SUBAPPLICATION SwitchPicCol_5_2 (* Bild- und Farbumschaltung für AUX-N und VT Objekte; 5 Zustände *)
  (* Standard: 61499-2 *)
  (* Version 1.1, 2026-04-09, Christoph Behr, HR Agrartechnik, Inits verbunden und REQ angeschlossen *)
  (* Version 1.0, 2025-06-12, franz, Meisterschulen am Ostbahnhof *)
  PACKAGE MyLib::sys;
  IMPORT logiBUS::utils::sequence::schieber::SchieberAuxInStruct;
  IMPORT logiBUS::utils::sequence::schieber::const::iSTATES::Unknown;
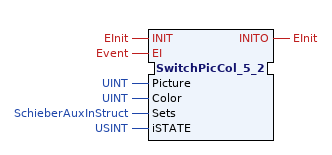
  EVENT_INPUT
    INIT : EInit; (* Initialization Request *)
    EI;
  END_EVENT
  EVENT_OUTPUT
    INITO : EInit; (* Initialization Confirm *)
  END_EVENT
  VAR_INPUT
    Picture : UINT; (* Object ID of the ObjectPointer to the Picture *)
    Color : UINT; (* Object ID of the AuxFunction *)
    Sets : logiBUS::utils::sequence::schieber::SchieberAuxInStruct;
    iSTATE : USINT := Unknown;
  END_VAR
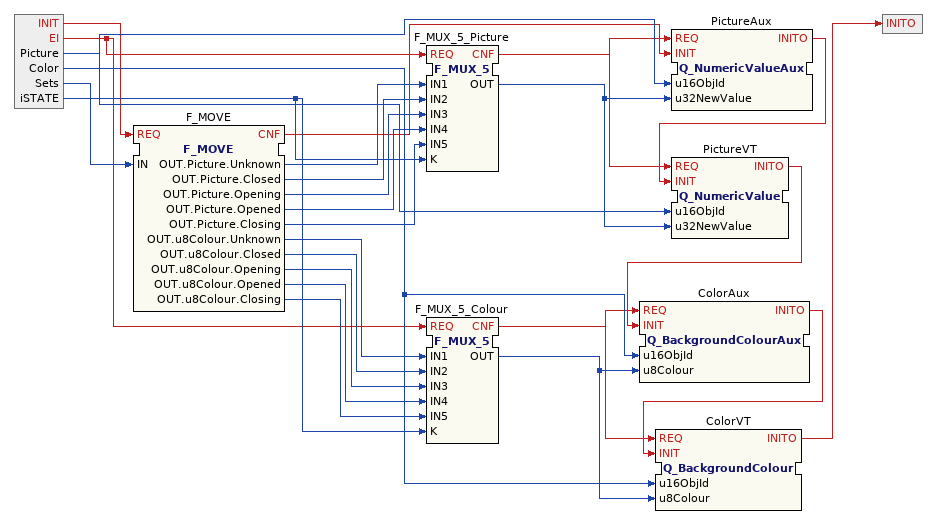
  FBS
    PictureVT : isobus::UT::Q::Q_NumericValue;
    ColorAux : isobus::UT::Q::Q_BackgroundColourAux;
    PictureAux : isobus::UT::Q::Q_NumericValueAux;
    ColorVT : isobus::UT::Q::Q_BackgroundColour;
    F_MOVE : iec61131::selection::F_MOVE; {SET_ATTRIBUTE(DataType, logiBUS::utils::sequence::schieber::SchieberAuxInStruct)}
    F_MUX_5_Picture : iec61131::selection::F_MUX_5;
    F_MUX_5_Colour : iec61131::selection::F_MUX_5;
  END_FBS
  EVENT_CONNECTIONS
    F_MUX_5_Picture.CNF TO PictureAux.REQ;
    F_MUX_5_Picture.CNF TO PictureVT.REQ;
    F_MUX_5_Colour.CNF TO ColorAux.REQ;
    F_MUX_5_Colour.CNF TO ColorVT.REQ;
    EI TO F_MUX_5_Picture.REQ;
    EI TO F_MUX_5_Colour.REQ;
    INIT TO F_MOVE.REQ;
    F_MOVE.CNF TO PictureAux.INIT;
    PictureAux.INITO TO PictureVT.INIT;
    PictureVT.INITO TO ColorAux.INIT;
    ColorAux.INITO TO ColorVT.INIT;
    ColorVT.INITO TO INITO;
  END_CONNECTIONS
  DATA_CONNECTIONS
    Color TO ColorAux.u16ObjId;
    Color TO ColorVT.u16ObjId;
    Picture TO PictureAux.u16ObjId;
    Picture TO PictureVT.u16ObjId;
    Sets TO F_MOVE.IN;
    F_MOVE.OUT.Picture.Unknown TO F_MUX_5_Picture.IN1;
    F_MOVE.OUT.Picture.Closed TO F_MUX_5_Picture.IN2;
    F_MOVE.OUT.Picture.Opening TO F_MUX_5_Picture.IN3;
    F_MOVE.OUT.Picture.Opened TO F_MUX_5_Picture.IN4;
    F_MOVE.OUT.Picture.Closing TO F_MUX_5_Picture.IN5;
    F_MOVE.OUT.u8Colour.Unknown TO F_MUX_5_Colour.IN1;
    F_MOVE.OUT.u8Colour.Closed TO F_MUX_5_Colour.IN2;
    F_MOVE.OUT.u8Colour.Opening TO F_MUX_5_Colour.IN3;
    F_MOVE.OUT.u8Colour.Opened TO F_MUX_5_Colour.IN4;
    F_MOVE.OUT.u8Colour.Closing TO F_MUX_5_Colour.IN5;
    F_MUX_5_Colour.OUT TO ColorAux.u8Colour;
    F_MUX_5_Colour.OUT TO ColorVT.u8Colour;
    F_MUX_5_Picture.OUT TO PictureAux.u32NewValue;
    F_MUX_5_Picture.OUT TO PictureVT.u32NewValue;
    iSTATE TO F_MUX_5_Picture.K;
    iSTATE TO F_MUX_5_Colour.K;
  END_CONNECTIONS
END_SUBAPPLICATION
